{attribute 'qualified_only'}
{attribute 'strict'}
TYPE
    E_DataFrom :
    (
        Local := 0,
        Remote := 1
    );
END_TYPE

(* stored: Version 1.1.0.1, ProductVersion 3.1.4024.13
   DUT E_DataFrom: Id {b8a47697-49a8-4404-b742-c5530b77b378} *)
